TYPE structAlarm :
STRUCT
	xAlarmIN	:	BOOL;	//Alarm Trigger
	xAlarmOFF	:	BOOL;	//Alarm übersteuert (wird nicht ausgelöst)
	xAlarmSAVE	:	BOOL;	//Alarm gespeichert (muss quittiert werden)
	xAlarmQUIT	:	BOOL;	//Alarm quittieren
	xAlarmOUT	:	BOOL;	//Alarm aktiv
	tAlarmVERZ	:	TIME;	//Alarmverzögerung
	sAlarmText	:	STRING;	//Alarmtext
	bAlarmNr	:	BYTE;	//Zusatztext #
END_STRUCT
END_TYPE

(* stored: Version 1.1.0.1, ProductVersion 3.1.4022.18
   DUT structAlarm: Id {1e9ea97c-e62d-4967-92d0-b39c1db2853d} *)
